RoboDK station: scene.rdk

Station scene (saved by RoboDK 5.9.0). Poses are relative to the parent item; angles as X-Y-Z fixed-axis rotations.
  - frame SPOT at (0, 0, 0) mm
    - frame Main_Origin at (-1867, -3409, 321) mm, rotated rx 15.91 ry -88.27 rz -124.22 deg
    - frame Secondary_Origin at (2176, -781, 346) mm, rotated rx 72.89 ry -88.78 rz -100.78 deg
